// TIA Portal V16 export
// export: Created 2024-05-11T02:56:23.0791915Z, ExportSetting WithDefaults, DisplayName Totally Integrated Automation Portal, DisplayVersion V16, DisplayName TIA Portal Version Control Interface, DisplayVersion V16, DisplayName TIA Portal Openness, DisplayVersion V16, DisplayName STEP 7 Professional, DisplayVersion V16, DisplayName STEP 7 Safety, DisplayVersion V16, DisplayName WinCC Professional, DisplayVersion V16
VAR_GLOBAL   // PLC tag table "100固定地址变量表"
   ManAutoPB AT %I1.0 : Bool;   // 手动/自动   {ExternalVisible false}
   StartPB AT %I1.1 : Bool;   // 启动(固定)
   StopPB AT %I1.2 : Bool;   // 停止(固定)
   RestPB AT %I1.3 : Bool;   // 复位(固定)
   EM_PB AT %I1.4 : Bool;   // 急停(固定)
   Buzzer AT %Q0.4 : Bool;   // 蜂鸣器Bz
   R_LED AT %Q0.5 : Bool;   // 三色灯<红>
   G_LED AT %Q0.6 : Bool;   // 三色灯<绿>
   Y_LED AT %Q0.7 : Bool;   // 三色灯<黄>
   Auto_LED AT %Q1.0 : Bool;   // 自动灯
   Clock_Byte AT %MB0 : Byte;
   System_Byte AT %MB1 : Byte;
   "0.1s时钟" AT %M0.0 : Bool;
   "0.2s时钟" AT %M0.1 : Bool;
   "0.4s时钟" AT %M0.2 : Bool;
   "0.5s时钟" AT %M0.3 : Bool;
   "0.8s时钟" AT %M0.4 : Bool;
   "1.0s时钟" AT %M0.5 : Bool;
   "1.6s时钟" AT %M0.6 : Bool;
   "2s时钟" AT %M0.7 : Bool;
   初始 AT %M1.0 : Bool;
   DiagStatusUpdate AT %M1.1 : Bool;
   常ON AT %M1.2 : Bool;
   常OFF AT %M1.3 : Bool;
   Int_M AT %M2.0 : Bool;   // xx
   Init_2s AT %M2.1 : Bool;   // 初始2s
   Run_2s AT %M2.2 : Bool;   // 运行2s
   Run_3s AT %M2.3 : Bool;   // 运行3s
   Run_4s AT %M2.4 : Bool;   // 运行4s
   AutoStep_P AT %M2.6 : Bool;   // 单步脉冲
   Fault_Rest AT %M2.7 : Bool;   // 故障复位
   Com_EMO AT %M3.0 : Bool;   // 总急停
   Com_SLC AT %M3.1 : Bool;   // 总光栅
   Com_DSW AT %M3.2 : Bool;   // 总门SW
   Com_OtherSafe AT %M3.3 : Bool;   // 其它安全
   Com_AirALM AT %M3.4 : Bool;   // 总气压
   AllFaults AT %M6.0 : Bool;   // 全部故障
   AllALM AT %M6.1 : Bool;   // 严重报警
   AllERR AT %M6.2 : Bool;   // 错误报警
   AllPoint AT %M6.3 : Bool;   // 提示信息
   FaultBuzzer AT %M6.7 : Bool;   // 蜂鸣器
   ManMode AT %M100.0 : Bool;   // 手动(固定)
   InitPB_All AT %M105.0 : Bool;   // 全初始化
   SN1_InitPB AT %M110.0 : Bool;   // SN1初始化
   SN1_Initial AT %M110.3 : Bool;   // SN1初始位
   SN1_InitStart AT %M110.4 : Bool;   // SN1初始化开始
   SN1_InitEnd AT %M110.5 : Bool;   // SN1初始化结束
   SN2_InitPB AT %M112.0 : Bool;   // SN2初始化
   SN2_Initial AT %M112.3 : Bool;   // SN2初始位
   SN2_InitStart AT %M112.4 : Bool;   // SN2初始化开始
   SN2_InitEnd AT %M112.5 : Bool;   // SN2初始化结束
   SN3_InitPB AT %M114.0 : Bool;   // SN3初始化
   SN3_Initial AT %M114.3 : Bool;   // SN3初始位
   SN3_InitStart AT %M114.4 : Bool;   // SN3初始化开始
   SN3_InitEnd AT %M114.5 : Bool;   // SN3初始化结束
   SN4_InitPB AT %M116.0 : Bool;   // SN4初始化
   SN4_Initial AT %M116.3 : Bool;   // SN4初始位
   SN4_InitStart AT %M116.4 : Bool;   // SN4初始化开始
   SN4_InitEnd AT %M116.5 : Bool;   // SN4初始化结束
   SN5_InitPB AT %M118.0 : Bool;   // SN5初始化
   SN5_Initial AT %M118.3 : Bool;   // SN5初始位
   SN5_InitStart AT %M118.4 : Bool;   // SN5初始化开始
   SN5_InitEnd AT %M118.5 : Bool;   // SN5初始化结束
   SN6_InitPB AT %M120.0 : Bool;   // SN6初始化
   SN6_Initial AT %M120.3 : Bool;   // SN6初始位
   SN6_InitStart AT %M120.4 : Bool;   // SN6初始化开始
   SN6_InitEnd AT %M120.5 : Bool;   // SN6初始化结束
   SN7_InitPB AT %M122.0 : Bool;   // SN7初始化
   SN7_Initial AT %M122.3 : Bool;   // SN7初始位
   SN7_InitStart AT %M122.4 : Bool;   // SN7初始化开始
   SN7_InitEnd AT %M122.5 : Bool;   // SN7初始化结束
   SN8_InitPB AT %M124.0 : Bool;   // SN8初始化
   SN8_Initial AT %M124.3 : Bool;   // SN8初始位
   SN8_InitStart AT %M124.4 : Bool;   // SN8初始化开始
   SN8_InitEnd AT %M124.5 : Bool;   // SN8初始化结束
   SN9_InitPB AT %M126.0 : Bool;   // SN9初始化
   SN9_Initial AT %M126.3 : Bool;   // SN9初始位
   SN9_InitStart AT %M126.4 : Bool;   // SN9初始化开始
   SN9_InitEnd AT %M126.5 : Bool;   // SN9初始化结束
   SN10_InitPB AT %M128.0 : Bool;   // SN10初始化
   SN10_Initial AT %M128.3 : Bool;   // SN10初始位
   SN10_InitStart AT %M128.4 : Bool;   // SN10初始化开始
   SN10_InitEnd AT %M128.5 : Bool;   // SN10初始化结束
   SN11_InitPB AT %M130.0 : Bool;   // SN11初始化
   SN11_Initial AT %M130.3 : Bool;   // SN11初始位
   SN11_InitStart AT %M130.4 : Bool;   // SN11初始化开始
   SN11_InitEnd AT %M130.5 : Bool;   // SN11初始化结束
   SN12_InitPB AT %M132.0 : Bool;   // SN12初始化
   SN12_Initial AT %M132.3 : Bool;   // SN12初始位
   SN12_InitStart AT %M132.4 : Bool;   // SN12初始化开始
   SN12_InitEnd AT %M132.5 : Bool;   // SN12初始化结束
   SN13_InitPB AT %M134.0 : Bool;   // SN13初始化
   SN13_Initial AT %M134.3 : Bool;   // SN13初始位
   SN13_InitStart AT %M134.4 : Bool;   // SN13初始化开始
   SN13_InitEnd AT %M134.5 : Bool;   // SN13初始化结束
   SN14_InitPB AT %M136.0 : Bool;   // SN14初始化
   SN14_Initial AT %M136.3 : Bool;   // SN14初始位
   SN14_InitStart AT %M136.4 : Bool;   // SN14初始化开始
   SN14_InitEnd AT %M136.5 : Bool;   // SN14初始化结束
   SN15_InitPB AT %M138.0 : Bool;   // SN15初始化
   SN15_Initial AT %M138.3 : Bool;   // SN15初始位
   SN15_InitStart AT %M138.4 : Bool;   // SN15初始化开始
   SN15_InitEnd AT %M138.5 : Bool;   // SN15初始化结束
   SN16_InitPB AT %M140.0 : Bool;   // SN16初始化
   SN16_Initial AT %M140.3 : Bool;   // SN16初始位
   SN16_InitStart AT %M140.4 : Bool;   // SN16初始化开始
   SN16_InitEnd AT %M140.5 : Bool;   // SN16初始化结束
   SN17_InitPB AT %M142.0 : Bool;   // SN17初始化
   SN17_Initial AT %M142.3 : Bool;   // SN17初始位
   SN17_InitStart AT %M142.4 : Bool;   // SN17初始化开始
   SN17_InitEnd AT %M142.5 : Bool;   // SN17初始化结束
   SN18_InitPB AT %M144.0 : Bool;   // SN18初始化
   SN18_Initial AT %M144.3 : Bool;   // SN18初始位
   SN18_InitStart AT %M144.4 : Bool;   // SN18初始化开始
   SN18_InitEnd AT %M144.5 : Bool;   // SN18初始化结束
   SN19_InitPB AT %M146.0 : Bool;   // SN19初始化
   SN19_Initial AT %M146.3 : Bool;   // SN19初始位
   SN19_InitStart AT %M146.4 : Bool;   // SN19初始化开始
   SN19_InitEnd AT %M146.5 : Bool;   // SN19初始化结束
   SN20_InitPB AT %M148.0 : Bool;   // SN20初始化
   SN20_Initial AT %M148.3 : Bool;   // SN20初始位
   SN20_InitStart AT %M148.4 : Bool;   // SN20初始化开始
   SN20_InitEnd AT %M148.5 : Bool;   // SN20初始化结束
   AutoMode AT %M150.0 : Bool;   // 自动模式
   AutoCont_Cut AT %M150.1 : Bool;   // 自动条件
   AutoPB_OFF AT %M150.2 : Bool;   // 自动OFF
   AutoStopReq AT %M150.3 : Bool;   // 自动停止要求
   Auto AT %M150.4 : Bool;   // 自动中
   InitPos AT %M150.5 : Bool;   // 初始位置
   AutoStop AT %M150.6 : Bool;   // 自动停止
   AlarmStop AT %M151.0 : Bool;   // 故障停止
   ErrorStop AT %M151.1 : Bool;   // 错误停止
   "SN1_Step(入口)" AT %MW200 : Int;   // SN1流程步
   "SN1_Start(入口)" AT %M250.0 : Bool;   // SN1开始
   "SN1_End(入口)" AT %M250.1 : Bool;   // SN1结束
   "SN1_搬入(入口)" AT %M250.2 : Bool;
   "SN1_搬出(入口)" AT %M250.3 : Bool;
   "SN2_Step(出口)" AT %MW202 : Int;   // SN2流程步
   "SN2_Start(出口)" AT %M252.0 : Bool;   // SN2开始
   "SN2_End(出口)" AT %M252.1 : Bool;   // SN2结束
   "SN2_搬入(出口)" AT %M252.2 : Bool;
   "SN2_搬出(出口)" AT %M252.3 : Bool;
   "SN3_Step(ST01上)" AT %MW204 : Int;   // SN3流程步
   "SN3_Start(ST01上)" AT %M254.0 : Bool;   // SN3开始
   "SN3_End(ST01上)" AT %M254.1 : Bool;   // SN3结束
   "SN3_搬入(ST01上)" AT %M254.2 : Bool;
   "SN3_搬出(ST01上)" AT %M254.3 : Bool;
   ST01放行标志 AT %M254.7 : Bool;
   "SN4_Step(ST02上)" AT %MW206 : Int;   // SN4流程步
   "SN4_Start(ST02上)" AT %M256.0 : Bool;   // SN4开始
   "SN4_End(ST02上)" AT %M256.1 : Bool;   // SN4结束
   "SN4_搬入(ST02上)" AT %M256.2 : Bool;
   "SN4_搬出(ST02上)" AT %M256.3 : Bool;
   ST02放行标志 AT %M256.7 : Bool;
   "SN5_Step(ST03上)" AT %MW208 : Int;   // SN5流程步
   "SN5_Start(ST03上)" AT %M258.0 : Bool;   // SN5开始
   "SN5_End(ST03上)" AT %M258.1 : Bool;   // SN5结束
   "SN5_搬入(ST03上)" AT %M258.2 : Bool;
   "SN5_搬出(ST03上)" AT %M258.3 : Bool;
   ST03放行标志 AT %M258.7 : Bool;
   "SN6_Step(ST04上)" AT %MW214 : Int;   // SN6流程步
   "SN6_Start(ST04上)" AT %M260.0 : Bool;   // SN6开始
   "SN6_End(ST04上)" AT %M260.1 : Bool;   // SN6结束
   "SN6_搬入(ST04上)" AT %M260.2 : Bool;
   "SN6_搬出(ST04上)" AT %M260.3 : Bool;
   ST04放行标志 AT %M260.7 : Bool;
   "SN7_Step(ST05上)" AT %MW216 : Int;   // SN7流程步
   "SN7_Start(ST05上)" AT %M262.0 : Bool;   // SN7开始
   "SN7_End(ST05上)" AT %M262.1 : Bool;   // SN7结束
   "SN7_搬入(ST05上)" AT %M262.2 : Bool;
   "SN7_搬出(ST05上)" AT %M262.3 : Bool;
   ST05放行标志 AT %M262.7 : Bool;
   "SN8_Step(ST06上)" AT %MW218 : Int;   // SN8流程步
   "SN8_Start(ST06上)" AT %M264.0 : Bool;   // SN8开始
   "SN8_End(ST06上)" AT %M264.1 : Bool;   // SN8结束
   "SN8_搬入(ST06上)" AT %M264.2 : Bool;
   "SN8_搬出(ST06上)" AT %M264.3 : Bool;
   ST06放行标志 AT %M264.7 : Bool;
   "SN9_Step(ST07上)" AT %MW222 : Int;   // SN9流程步
   "SN9_Start(ST07上)" AT %M265.0 : Bool;   // SN9开始
   "SN9_End(ST07上)" AT %M266.1 : Bool;   // SN9结束
   "SN9_搬入(ST07上)" AT %M266.2 : Bool;
   "SN9_搬出(ST07上)" AT %M266.3 : Bool;
   ST07放行标志 AT %M266.7 : Bool;
   "SN10_Step(ST08上)" AT %MW224 : Int;   // SN10流程步
   "SN10_Start(ST08上)" AT %M268.0 : Bool;   // SN10开始
   "SN10_End(ST08上)" AT %M268.1 : Bool;   // SN10结束
   "SN10_搬入(ST08上)" AT %M268.2 : Bool;
   "SN10_搬出(ST08上)" AT %M268.3 : Bool;
   ST08放行标志 AT %M268.7 : Bool;
   "SN11_Step(ST09上)" AT %MW226 : Int;   // SN11流程步
   "SN11_Start(ST09上)" AT %M270.0 : Bool;   // SN11开始
   "SN11_End(ST09上)" AT %M270.1 : Bool;   // SN11结束
   "SN11_搬入(ST09上)" AT %M270.2 : Bool;
   "SN11_搬出(ST09上)" AT %M270.3 : Bool;
   ST09放行标志 AT %M270.7 : Bool;
   "SN12_Step(ST10上)" AT %MW228 : Int;   // SN12流程步
   "SN12_Start(ST10上)" AT %M272.0 : Bool;   // SN12开始
   "SN12_End(ST10上)" AT %M272.1 : Bool;   // SN12结束
   "SN12_搬入(ST10上)" AT %M272.2 : Bool;
   "SN12_搬出(ST10上)" AT %M272.3 : Bool;
   ST10放行标志 AT %M272.7 : Bool;
   "SN13_Step(ST11上)" AT %MW230 : Int;   // SN13流程步
   "SN13_Start(ST11上)" AT %M274.0 : Bool;   // SN13开始
   "SN13_End(ST11上)" AT %M274.1 : Bool;   // SN13结束
   "SN13_搬入(ST11上)" AT %M274.2 : Bool;
   "SN13_搬出(ST11上)" AT %M274.3 : Bool;
   ST11放行标志 AT %M274.7 : Bool;
   "SN14_Step(ST12上)" AT %MW232 : Int;   // SN14流程步
   "SN14_Start(ST12上)" AT %M276.0 : Bool;   // SN14开始
   "SN14_End(ST12上)" AT %M276.1 : Bool;   // SN14结束
   "SN14_搬入(ST12上)" AT %M276.2 : Bool;
   "SN14_搬出(ST12上)" AT %M276.3 : Bool;
   ST12放行标志 AT %M276.7 : Bool;
   "SN15_Step(ST03下)" AT %MW234 : Int;   // SN15流程步
   SN15_Start AT %M278.0 : Bool;   // SN15开始
   SN15_End AT %M278.1 : Bool;   // SN15结束
   SN15_搬入 AT %M278.2 : Bool;
   SN15_搬出 AT %M278.3 : Bool;
   "SN16_Step(ST02下)" AT %MW236 : Int;   // SN16流程步
   SN16_Start AT %M280.0 : Bool;   // SN16开始
   SN16_End AT %M280.1 : Bool;   // SN16结束
   SN16_搬入 AT %M280.2 : Bool;
   SN16_搬出 AT %M280.3 : Bool;
   "SN17_Step(ST01下)" AT %MW238 : Int;   // SN17流程步
   SN17_Start AT %M282.0 : Bool;   // SN17开始
   SN17_End AT %M282.1 : Bool;   // SN17结束
   SN17_搬入 AT %M282.2 : Bool;
   SN17_搬出 AT %M282.3 : Bool;
   SN18_Step AT %MW240 : Int;   // SN18流程步
   SN18_Start AT %M284.0 : Bool;   // SN18开始
   SN18_End AT %M284.1 : Bool;   // SN18结束
   SN18_搬入 AT %M284.2 : Bool;
   SN18_搬出 AT %M284.3 : Bool;
   SN19_Step AT %MW242 : Int;   // SN19流程步
   SN19_Start AT %M286.0 : Bool;   // SN19开始
   SN19_End AT %M286.1 : Bool;   // SN19结束
   SN19_搬入 AT %M286.2 : Bool;
   SN19_搬出 AT %M286.3 : Bool;
   SN20_Step AT %MW244 : Int;   // SN20流程步
   SN20_Start AT %M288.0 : Bool;   // SN20开始
   SN20_End AT %M288.1 : Bool;   // SN20结束
   SN20_搬入 AT %M288.2 : Bool;
   SN20_搬出 AT %M288.3 : Bool;
   AutoStep AT %M600.0 : Bool;   // 自动单步
   LampTest AT %M600.1 : Bool;   // 灯测试
   Durable AT %M600.2 : Bool;   // 耐久模式
   ST01屏蔽 AT %M650.0 : Bool;
   ST02屏蔽 AT %M650.1 : Bool;
   ST03屏蔽 AT %M650.2 : Bool;
   ST04屏蔽 AT %M650.3 : Bool;
   ST05屏蔽 AT %M650.4 : Bool;
   ST06屏蔽 AT %M650.5 : Bool;
   ST07屏蔽 AT %M650.6 : Bool;
   ST08屏蔽 AT %M650.7 : Bool;
   ST09屏蔽 AT %M651.0 : Bool;
   ST10屏蔽 AT %M651.1 : Bool;
   ST11屏蔽 AT %M651.2 : Bool;
   ST12屏蔽 AT %M651.3 : Bool;
   ST13屏蔽 AT %M651.4 : Bool;
   ST14屏蔽 AT %M651.5 : Bool;
   ST15屏蔽 AT %M651.6 : Bool;
   ST16屏蔽 AT %M651.7 : Bool;
   ST17屏蔽 AT %M652.0 : Bool;
   ST18屏蔽 AT %M652.1 : Bool;
   ST19屏蔽 AT %M652.2 : Bool;
   ST20屏蔽 AT %M652.3 : Bool;
   生产数量清零 AT %M695.0 : Bool;
   累计数量清零 AT %M695.1 : Bool;
END_VAR
